FUNCTION_BLOCK FB_SerialScale EXTENDS FB_ComponentBase IMPLEMENTS I_Scale
VAR
	_InSimulation : BOOL;
END_VAR

//{warning 'Add method implementation '}
METHOD CyclicLogic
IF _InSimulation THEN
	CyclicSimulate();
ELSE
	;
END_IF
END_METHOD

METHOD CyclicSimulate
VAR_INPUT
END_VAR
END_METHOD

PROPERTY InSimulation : BOOL
GET
InSimulation := _InSimulation;
END_GET
SET
_InSimulation := InSimulation;
END_SET
END_PROPERTY

{warning 'Add method implementation '}
METHOD Tare
END_METHOD

{warning 'Add property implementation'}
PROPERTY Weight : LREAL
GET
END_GET
SET
END_SET
END_PROPERTY

END_FUNCTION_BLOCK

(* stored: Version 1.1.0.1
   POU FB_SerialScale: Id {d17ba426-4188-4e8b-96c7-883096957677}, SpecialFunc None
   Method CyclicLogic: Id {cf7b4cb0-8c33-4ff6-bf09-d5dd5790293c}
   Method CyclicSimulate: Id {1951040f-be21-4749-8f68-af3910f5ef3f}
   Property InSimulation: Id {3596a00c-3fdf-46e1-be99-df220d6c569e}
   Get Get: Id {8680dcab-99b9-4c55-95e3-07b4ce2e38fa}
   Set Set: Id {66cbb3ba-0518-4383-8e5d-a853cfec42c2}
   Method Tare: Id {2ef36671-ceaf-4d0a-82f6-ee497fc7992e}
   Property Weight: Id {3185b20a-f881-4eda-8a69-d21813084103}
   Get Get: Id {172a951e-9461-476c-a497-759922d13dad}
   Set Set: Id {d1d405cb-4b6b-4c2e-b277-0a7cbb389bd6} *)
